(*
SPDX-FileCopyrightText: © 2026 Oleksandr Tiutyk <trofimich@gmail.com>
SPDX-License-Identifier: MIT
License: https://opensource.org/license/mit
*)

INTERFACE IExceptionHandlingPolicy EXTENDS IObject

METHOD HandleException : EXCEPTION_REACTION
VAR_INPUT
	exception : IReadOnlyException;
	handlingObject : IObject;
END_VAR
VAR_IN_OUT CONSTANT
	failedMethodName : STRING(255);
END_VAR
END_METHOD

END_INTERFACE

(* stored: Version 1.1.0.1
   Itf IExceptionHandlingPolicy: Id {d50dbbea-981a-44d1-80f2-547a2b018dd7}
   Method HandleException: Id {4d297766-4165-4ad2-b0ec-d1c1753b7530} *)
